TYPE E_VGC :
(

	Vented,
	Vacuum,
	ERR_DiffPress,
	ERR_LostVac

);
END_TYPE

(* stored: Version 1.1.0.1, ProductVersion 3.1.0.24
   DUT E_VGC: Id {e141839c-aa77-413d-8cbc-038cd47aa3b1} *)
